{attribute addProperty BoxType "EL5001-0000-1017"}
{attribute addProperty Id "SSI_InputsAT %I*SSI_Inputs_F7D238D14860WcStateAT %I*WcState_98A4DF7520.250InfoDataAT %I*InfoData_BC63D37F80100"}
{attribute addProperty CRC "2564453052"}
{attribute addProperty SizeInBites "130"}
{attribute addProperty SizeInBytes "16.25"}
TYPE EL5001_2283773F :
STRUCT
	{attribute addProperty Name "SSI_Inputs"}
	SSI_Inputs : SSI_Inputs_F7D238D1;
	{attribute addProperty Name "WcState"}
	WcState : WcState_98A4DF75;
	{attribute addProperty Name "InfoData"}
	InfoData : InfoData_BC63D37F;
END_STRUCT
END_TYPE

(* stored: Version 1.2.0.0, ProductVersion 3.1.4024.9
   DUT EL5001_2283773F: Id {a602b3f5-a527-469b-80d6-8528cabf0b79} *)
